// TwinCAT 3 PLC project Practice_3
// ProgramVersion: 3.1.4024.0
// libraries:
//   Tc2_Standard, * (Beckhoff Automation GmbH)
//   Tc2_System, * (Beckhoff Automation GmbH)
//   Tc3_Module, * (Beckhoff Automation GmbH)
// project tree:
//   / PlcTask.TcTTO
//   POUs/ MAIN.TcPOU
// (motion and I/O tree: see PLC project practice_1)
// real-time tasks:
//   TASK PlcTask: cycle T#10ms, priority 20, ADS port 350
//   TASK PlcTask1: cycle T#10ms, priority 21, ADS port 351
//   TASK PlcTask2: cycle T#10ms, priority 22, ADS port 352

CONFIGURATION Practice_3
    RESOURCE PLC ON TwinCAT3
        TASK PlcTask(INTERVAL := T#10ms, PRIORITY := 22);
        PROGRAM MAIN WITH PlcTask : MAIN;
    END_RESOURCE
END_CONFIGURATION

// ---- POUs/MAIN.TcPOU
PROGRAM MAIN
VAR
	sInputString : STRING;
END_VAR

END_PROGRAM
